Staubli VAL3: Main.pgx

program Main()
  local num l_nKey
begin
  //
 do
    call Refresh()
    call RefreshList()
    call user:setList("路径",sFileList,bUserRefresh,bListRefresh,nSelected,sItem,l_nKey)
    bUserRefresh=false
    bListRefresh=false
    call MainKey(l_nKey)
    delay(0)
  until bExit

end
